FUNCTION_BLOCK W2W3 (* Basic Function Block Type *)
  (* Standard: 61499-2 *)
  (* Version 0.0, 9/24/2018, dmidro, nxtControl GmbH, Template *)
  PACKAGE Main;
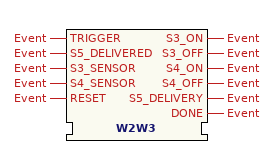
  EVENT_INPUT
    TRIGGER;
    S5_DELIVERED;
    S3_SENSOR;
    S4_SENSOR;
    RESET;
  END_EVENT
  EVENT_OUTPUT
    S3_ON;
    S3_OFF;
    S4_ON;
    S4_OFF;
    S5_DELIVERY;
    DONE;
  END_EVENT
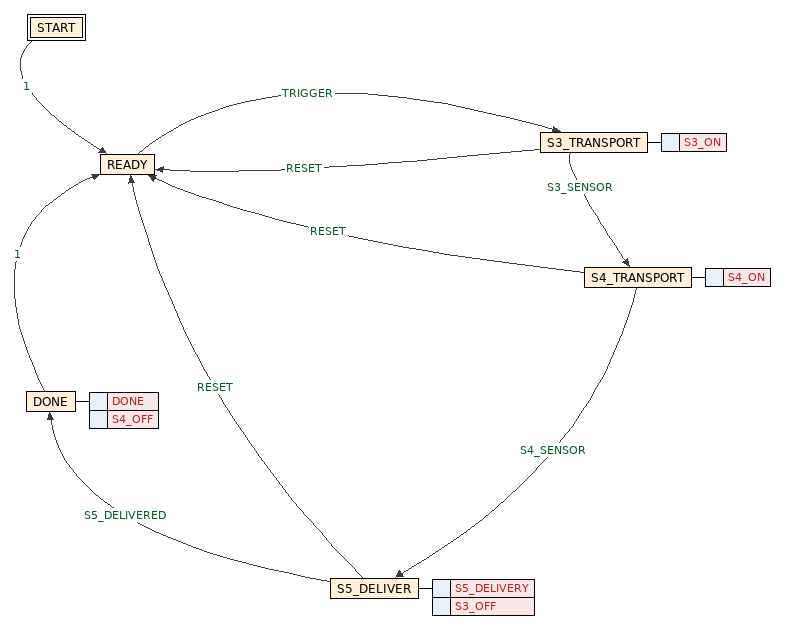
  EC_STATES
    START; (* Initial State *)
    S3_TRANSPORT : -> S3_ON;
    S4_TRANSPORT : -> S4_ON;
    S5_DELIVER : -> S5_DELIVERY, -> S3_OFF;
    DONE : -> DONE, -> S4_OFF;
    READY;
  END_STATES
  EC_TRANSITIONS
    START TO READY := 1;
    S3_TRANSPORT TO S4_TRANSPORT := S3_SENSOR;
    S5_DELIVER TO DONE := S5_DELIVERED;
    READY TO S3_TRANSPORT := TRIGGER;
    DONE TO READY := 1;
    S4_TRANSPORT TO S5_DELIVER := S4_SENSOR;
    S3_TRANSPORT TO READY := RESET;
    S4_TRANSPORT TO READY := RESET;
    S5_DELIVER TO READY := RESET;
  END_TRANSITIONS
  ALGORITHM INIT IN ST: (* Initialization algorithm *)
;
  END_ALGORITHM
  ALGORITHM REQ IN ST: (* Normally executed algorithm *)
;
  END_ALGORITHM
END_FUNCTION_BLOCK
